// TIA Portal project "helloWorld" (V14)

(* hardware
DEVICE "S71500/ET200MP station_1"  S7-1500 station
   slot 0: "导轨_0"  Rack  6ES7 590-1***0-0AA0
   slot 1: "PLC_1"  CPU 1511-1 PN  6ES7 511-1AK01-0AB0  V1.8
      slot 3: "CPU 显示_1"  6ES7591-1AA00-0AA0
DEVICE "PC-System_1"  SIMATIC PC station
   slot 0: "SIMATIC PC station"  Rail  SIMATIC PC-Station  V1.0
      slot 125: "Stationmanager"  Station_Manager  V6.0.4
   slot 1: "HMI_RT_1"  WinCC RT Advanced  6AV2 104-0xxxx-xxxx  14.0.1.0
      slot 33792: "主机接口"  Host interface
   slot 2: "IE general_1"  IE General  IE_CP  V8.2.0
*)

// ===== PLC "PLC_1"  CPU 1511-1 PN =====

DATA_BLOCK "input"   // DB1
{ S7_Optimized_Access := 'FALSE' }
VERSION : 0.1
   VAR
      _1 : Bool;
      _2 : Bool;
      _3 : Bool;
      _4 : Bool;
      _5 : Bool;
      _6 : Bool;
      _7 : Bool;
      _8 : Bool;
      _9 : Bool;
      _10 : Bool;
      _11 : Bool;
      _12 : Bool;
      _13 : Bool;
      _14 : Bool;
      _15 : Bool;
      _16 : Bool;
      _17 : Bool;
      _18 : Bool;
      _19 : Bool;
      _20 : Bool;
      _21 : Bool;
      _22 : Bool;
      _23 : Bool;
      _24 : Bool;
      _25 : Bool;
      _26 : Bool;
      _27 : Bool;
      _28 : Bool;
      _29 : Bool;
      _30 : Bool;
      _31 : Bool;
      _32 : Bool;
      _33 : Bool;
      _34 : Bool;
      _35 : Bool;
      _36 : Bool;
      _37 : Word;
   END_VAR
BEGIN
END_DATA_BLOCK

DATA_BLOCK "output"   // DB2
{ S7_Optimized_Access := 'FALSE' }
VERSION : 0.1
   VAR
      _1 : Bool;
      _2 : Bool;
      _3 : Bool;
      _4 : Bool;
      _5 : Bool;
      _6 : Bool;
      _7 : Bool;
      _8 : Bool;
      _9 : Bool;
      _10 : Bool;
      _11 : Bool;
      _12 : Bool;
      _13 : Bool;
      _14 : Bool;
      _15 : Bool;
      _16 : Bool;
      _17 : Bool;
      _18 : Bool;
      _19 : Bool;
      _20 : Bool;
      _21 : Bool;
      _22 : Bool;
      _23 : Bool;
      _24 : Bool;
      _25 : Bool;
      _26 : Bool;
      _27 : Bool;
      _28 : Bool;
      _29 : Bool;
      _30 : Bool;
      _31 : Bool;
      _32 : Bool;
      _33 : Bool;
      _34 : Bool;
      _35 : Bool;
      _36 : Bool;
      _37 : Bool;
      _38 : Bool;
      _39 : Bool;
      _40 : Bool;
   END_VAR
BEGIN
END_DATA_BLOCK

ORGANIZATION_BLOCK "Main"   // OB1, LAD, ProgramCycle
TITLE = "Main Program Sweep (Cycle)"
{ S7_Optimized_Access := 'TRUE' }
VERSION : 0.1
   VAR_INPUT
      Initial_Call : Bool;   // Initial call of this OB
      Remanence : Bool;   // =True, if remanent data are available
   END_VAR
BEGIN

REGION Network 1
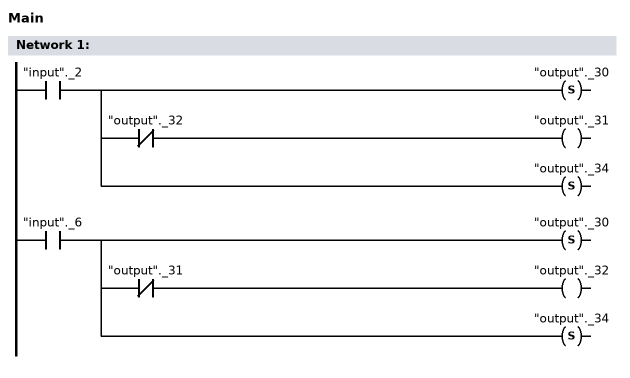
   RUNG wire#powerrail
      Contact( "input"._2 )
      wire#w1
      S_Coil( "output"._30 )
   END_RUNG
   RUNG wire#w1
      I_Contact( "output"._32 )
      Coil( "output"._31 )
   END_RUNG
   RUNG wire#w1
      S_Coil( "output"._34 )
   END_RUNG
   RUNG wire#powerrail
      Contact( "input"._6 )
      wire#w2
      S_Coil( "output"._30 )
   END_RUNG
   RUNG wire#w2
      I_Contact( "output"._31 )
      Coil( "output"._32 )
   END_RUNG
   RUNG wire#w2
      S_Coil( "output"._34 )
   END_RUNG
   // the same network as SCL:
   IF "input"._2 THEN "output"._30 := TRUE; END_IF;
   "output"._31 := "input"._2 AND NOT "output"._32;
   IF "input"._2 THEN "output"._34 := TRUE; END_IF;
   IF "input"._6 THEN "output"._30 := TRUE; END_IF;
   "output"._32 := "input"._6 AND NOT "output"._31;
   IF "input"._6 THEN "output"._34 := TRUE; END_IF;
END_REGION
END_ORGANIZATION_BLOCK

(* ===== HMI "HMI_RT_1" =====

screen "画面_1" 1024x768
   HTMLBrowser "HTML 浏览器_1" at 0,0 size 1024x767
*)